PROGRAM Regulation_Centrale_Hydro
VAR
	(*******************************************************************************************************************************************************)
	(******************************************** BLOC FONCTION POUR REGULATION PRESSION *******************************************)
	(*******************************************************************************************************************************************************)
	Regulation_Centrale_Hydraulique					: FB_Regulation_Centrale_Atos;

	(*******************************************************************************************************************************************************)
	(***************************************************** TRANSMITER DE PRESSION IFM IOLINK **********************************************)
	(*******************************************************************************************************************************************************)
	Capteur_Pression									: FB_IOLink_IFM_PV7000;
	No_Data_Pression_Huile							: BOOL;
	Over_Limite_Pression_Huile						: BOOL;


	(*******************************************************************************************************************************************************)
	(************************************** TRANSMITER DE NIVEAU ET TEMPERATURE ESLTI IOLINK ****************************************)
	(*******************************************************************************************************************************************************)
	FB_IOLink_ES_ESLTI: FB_IOLink_ES_ESLTI;
	Device_Ok: BOOL;
	Temp_Out_Of_Range: BOOL;
	Temperature_Celcius :LREAL;
	Pourcentage_Niveau :LREAL;

	(*******************************************************************************************************************************************************)
	(************************************************* VARIATEUR DE POMPE I550 MOTEC MURAL *********************************************)
	(*******************************************************************************************************************************************************)
	I550_Pompe_MoteC: FB_Var_LENZE_I550_Motec_Centrale_Atos;
	Accel											: UINT := 150;
	Decel											: UINT := 75;
	Consigne_Tr_Min_Centrale_Hydro					: INT;

	Demande_Basse_Pression							: BOOL;
	Niveau_OK										: BOOL;

	Voie_IOLink: BOOL;

END_VAR

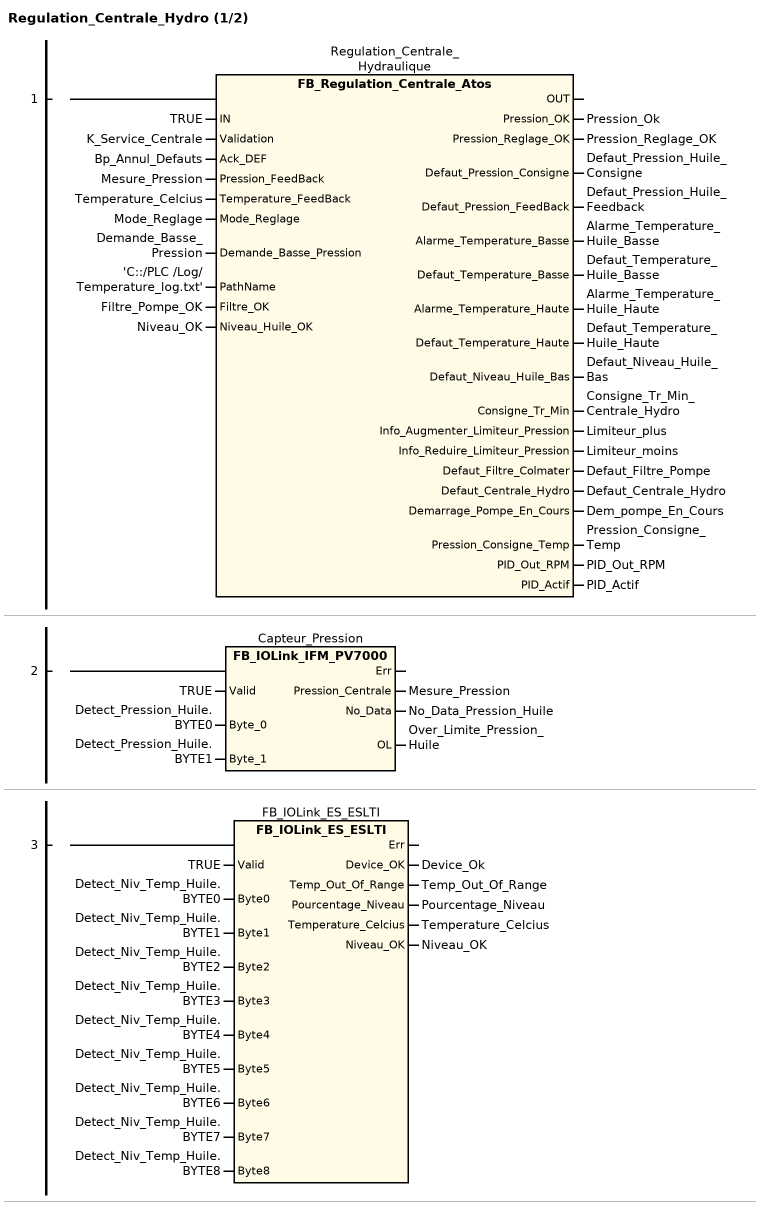
// NETWORK 1
Regulation_Centrale_Hydraulique(
    IN := TRUE,
    Validation := K_Service_Centrale,
    Ack_DEF := Bp_Annul_Defauts,
    Pression_FeedBack := Mesure_Pression,
    Temperature_FeedBack := Temperature_Celcius,
    Mode_Reglage := Mode_Reglage,
    Demande_Basse_Pression := Demande_Basse_Pression,
    PathName := 'C::/PLC /Log/Temperature_log.txt',
    Filtre_OK := Filtre_Pompe_OK,
    Niveau_Huile_OK := Niveau_OK,
    Pression_OK => Pression_Ok,
    Pression_Reglage_OK => Pression_Reglage_OK,
    Defaut_Pression_Consigne => Defaut_Pression_Huile_Consigne,
    Defaut_Pression_FeedBack => Defaut_Pression_Huile_Feedback,
    Alarme_Temperature_Basse => Alarme_Temperature_Huile_Basse,
    Defaut_Temperature_Basse => Defaut_Temperature_Huile_Basse,
    Alarme_Temperature_Haute => Alarme_Temperature_Huile_Haute,
    Defaut_Temperature_Haute => Defaut_Temperature_Huile_Haute,
    Defaut_Niveau_Huile_Bas => Defaut_Niveau_Huile_Bas,
    Consigne_Tr_Min => Consigne_Tr_Min_Centrale_Hydro,
    Info_Augmenter_Limiteur_Pression => Limiteur_plus,
    Info_Reduire_Limiteur_Pression => Limiteur_moins,
    Defaut_Filtre_Colmater => Defaut_Filtre_Pompe,
    Defaut_Centrale_Hydro => Defaut_Centrale_Hydro,
    Demarrage_Pompe_En_Cours => Dem_pompe_En_Cours,
    Pression_Consigne_Temp => Pression_Consigne_Temp,
    PID_Out_RPM => PID_Out_RPM,
    PID_Actif => PID_Actif); // FB_Regulation_Centrale_Atos

// NETWORK 2
Capteur_Pression(
    Valid := TRUE,
    Byte_0 := Detect_Pression_Huile.BYTE0,
    Byte_1 := Detect_Pression_Huile.BYTE1,
    Pression_Centrale => Mesure_Pression,
    No_Data => No_Data_Pression_Huile,
    OL => Over_Limite_Pression_Huile); // FB_IOLink_IFM_PV7000

// NETWORK 3
FB_IOLink_ES_ESLTI(
    Valid := TRUE,
    Byte0 := Detect_Niv_Temp_Huile.BYTE0,
    Byte1 := Detect_Niv_Temp_Huile.BYTE1,
    Byte2 := Detect_Niv_Temp_Huile.BYTE2,
    Byte3 := Detect_Niv_Temp_Huile.BYTE3,
    Byte4 := Detect_Niv_Temp_Huile.BYTE4,
    Byte5 := Detect_Niv_Temp_Huile.BYTE5,
    Byte6 := Detect_Niv_Temp_Huile.BYTE6,
    Byte7 := Detect_Niv_Temp_Huile.BYTE7,
    Byte8 := Detect_Niv_Temp_Huile.BYTE8,
    Device_OK => Device_Ok,
    Temp_Out_Of_Range => Temp_Out_Of_Range,
    Pourcentage_Niveau => Pourcentage_Niveau,
    Temperature_Celcius => Temperature_Celcius,
    Niveau_OK => Niveau_OK);

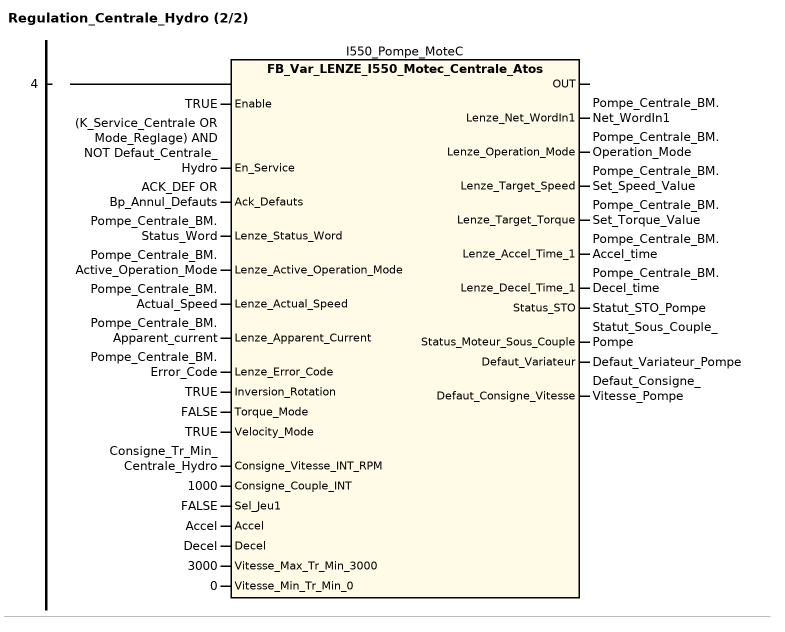
// NETWORK 4
I550_Pompe_MoteC(
    Enable := TRUE,
    En_Service := (K_Service_Centrale OR Mode_Reglage) AND NOT Defaut_Centrale_Hydro,
    Ack_Defauts := ACK_DEF OR Bp_Annul_Defauts,
    Lenze_Status_Word := Pompe_Centrale_BM.Status_Word,
    Lenze_Active_Operation_Mode := Pompe_Centrale_BM.Active_Operation_Mode,
    Lenze_Actual_Speed := Pompe_Centrale_BM.Actual_Speed,
    Lenze_Apparent_Current := Pompe_Centrale_BM.Apparent_current,
    Lenze_Error_Code := Pompe_Centrale_BM.Error_Code,
    Inversion_Rotation := TRUE,
    Torque_Mode := FALSE,
    Velocity_Mode := TRUE,
    Consigne_Vitesse_INT_RPM := Consigne_Tr_Min_Centrale_Hydro,
    Consigne_Couple_INT := 1000,
    Sel_Jeu1 := FALSE,
    Accel := Accel,
    Decel := Decel,
    Vitesse_Max_Tr_Min_3000 := 3000,
    Vitesse_Min_Tr_Min_0 := 0,
    Lenze_Net_WordIn1 => Pompe_Centrale_BM.Net_WordIn1,
    Lenze_Operation_Mode => Pompe_Centrale_BM.Operation_Mode,
    Lenze_Target_Speed => Pompe_Centrale_BM.Set_Speed_Value,
    Lenze_Target_Torque => Pompe_Centrale_BM.Set_Torque_Value,
    Lenze_Accel_Time_1 => Pompe_Centrale_BM.Accel_time,
    Lenze_Decel_Time_1 => Pompe_Centrale_BM.Decel_time,
    Status_STO => Statut_STO_Pompe,
    Status_Moteur_Sous_Couple => Statut_Sous_Couple_Pompe,
    Defaut_Variateur => Defaut_Variateur_Pompe,
    Defaut_Consigne_Vitesse => Defaut_Consigne_Vitesse_Pompe); // FB_Var_LENZE_I550_Motec_Centrale_Atos

END_PROGRAM

(* stored: Version 1.1.0.1
   POU Regulation_Centrale_Hydro: Id {3731edb0-7a20-4a36-ac4d-a94ee781f6e1}, SpecialFunc None *)
